Universal Robots URScript: move_lin_rel.script

def move_lin_rel():
    textmsg("Move_l via relative translation.")
    current_pos = get_actual_tcp_pose()
    offset_pose = p[{0}, {1}, {2}, 0.0, 0.0, 0.0]
    movel(pose_trans(current_pos, offset_pose), a = {3}, v = {4})
    textmsg("Done.")
end
